// TIA Portal project "Project1" (V18)
// sta je sad ovo koji k

(* hardware
DEVICE "S7-1200 station_1"  S7-1200 Station
   slot 0: "Rack_0"  S7-1200 Rack  Rack  V1.0
   slot 1: "PLC_1"  CPU 1211C AC/DC/Rly  6ES7 211-1BE40-0XB0  V4.6
*)

// ===== PLC "PLC_1"  CPU 1211C AC/DC/Rly =====

VAR_GLOBAL   // PLC tag table "Default tag table"
   "button1" AT %I0.0 : Bool;
   "green" AT %Q0.0 : Bool;
   "red" AT %Q0.1 : Bool;
   "yellow" AT %Q0.2 : Bool;
   "button2" AT %I0.1 : Bool;
   "limit_switch" AT %I0.2 : Bool;
   "reset" AT %I0.3 : Bool;
END_VAR

// folder: System blocks/Program resources

DATA_BLOCK "timer1"   // DB1
{ S7_Optimized_Access := 'TRUE' }
AUTHOR : Simatic
FAMILY : IEC
NAME : IEC_TMR
VERSION : 1.0
// stored: InstanceOfName IEC_TIMER
"IEC_TIMER"
BEGIN
END_DATA_BLOCK

DATA_BLOCK "timer2"   // DB2
{ S7_Optimized_Access := 'TRUE' }
AUTHOR : Simatic
FAMILY : IEC
NAME : IEC_TMR
VERSION : 1.0
// stored: InstanceOfName IEC_TIMER
"IEC_TIMER"
BEGIN
END_DATA_BLOCK

DATA_BLOCK "run_time"   // DB3
{ S7_Optimized_Access := 'TRUE' }
AUTHOR : Simatic
FAMILY : IEC
NAME : IEC_TMR
VERSION : 1.0
// stored: InstanceOfName IEC_TIMER
"IEC_TIMER"
BEGIN
END_DATA_BLOCK

// folder: (top level)

ORGANIZATION_BLOCK "Main"   // OB1, LAD, ProgramCycle
TITLE = "Main Program Sweep (Cycle)"
{ S7_Optimized_Access := 'TRUE' }
VERSION : 0.1
   VAR_INPUT
      Initial_Call : Bool;   // Initial call of this OB
      Remanence : Bool;   // =True, if remanent data are available
   END_VAR
   VAR_TEMP
      error : Bool;   // error state variable
      last_button1 : Bool;
      last_button2 : Bool;
      pressed1 : Bool;
      pressed2 : Bool;
      both_pressed : Bool;
      on : Bool;
   END_VAR
BEGIN

REGION Network 1
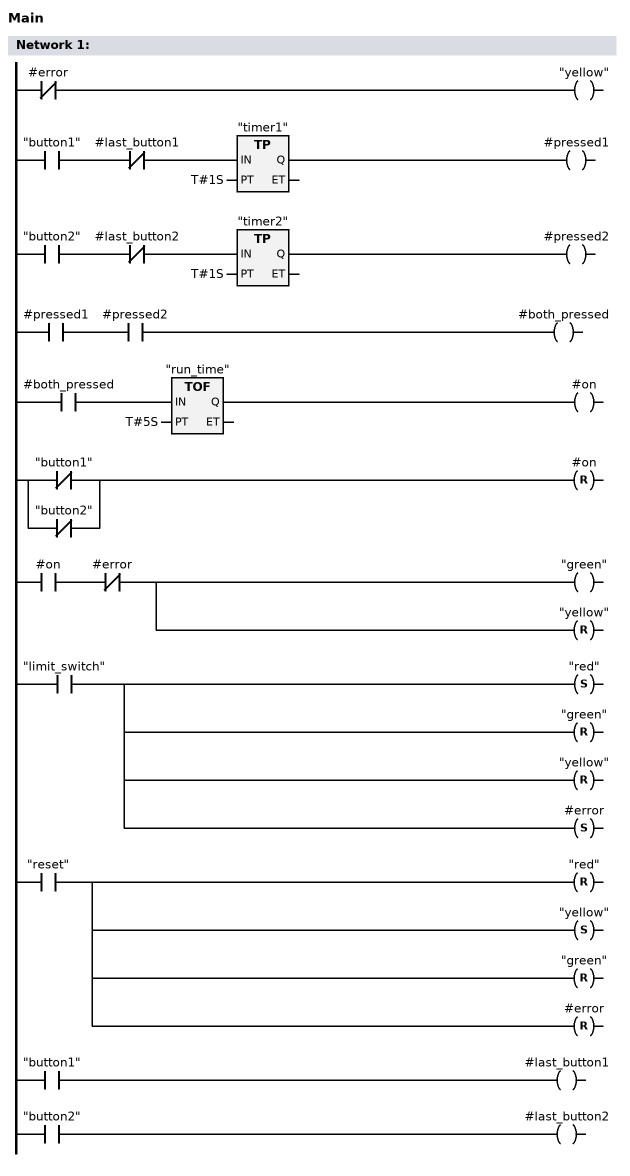
   "yellow" := NOT #error;
   "timer1".TP(IN := "button1" AND NOT #last_button1, PT := T#1S);
   #pressed1 := "timer1".Q;
   "timer2".TP(IN := "button2" AND NOT #last_button2, PT := T#1S);
   #pressed2 := "timer2".Q;
   #both_pressed := #pressed1 AND #pressed2;
   "run_time".TOF(IN := #both_pressed, PT := T#5S);
   #on := "run_time".Q;
   IF NOT "button1" OR NOT "button2" THEN #on := FALSE; END_IF;
   "green" := #on AND NOT #error;
   IF "green" THEN "yellow" := FALSE; END_IF;
   IF "limit_switch" THEN
       "red" := TRUE;
       "green" := FALSE;
       "yellow" := FALSE;
       #error := TRUE;
   END_IF;
   IF "reset" THEN
       "red" := FALSE;
       "yellow" := TRUE;
       "green" := FALSE;
       #error := FALSE;
   END_IF;
   #last_button1 := "button1";
   #last_button2 := "button2";
END_REGION
END_ORGANIZATION_BLOCK